// Mitsubishi GX Works2 project: a16   PLC: Q02/Q02H

PROGRAM MAIN
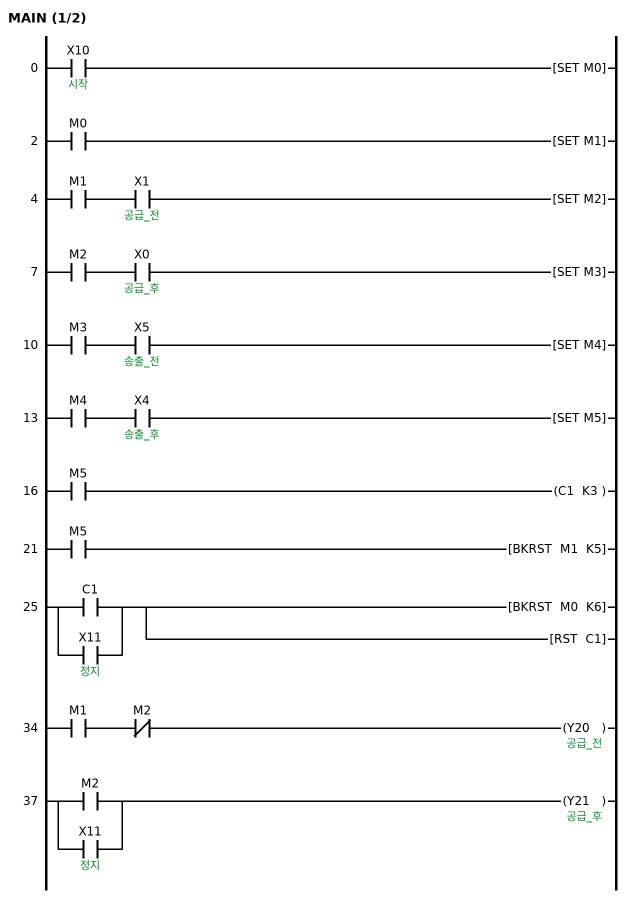
0     LD      X10  ; 시작
      SET     M0
2     LD      M0
      SET     M1
4     LD      M1
      AND     X1  ; 공급_전
      SET     M2
7     LD      M2
      AND     X0  ; 공급_후
      SET     M3
10    LD      M3
      AND     X5  ; 송출_전
      SET     M4
13    LD      M4
      AND     X4  ; 송출_후
      SET     M5
16    LD      M5
      OUT     C1 K3
21    LD      M5
      BKRST   M1 K5
25    LD      C1
      OR      X11  ; 정지
      BKRST   M0 K6
      RST     C1
34    LD      M1
      ANI     M2
      OUT     Y20  ; 공급_전
37    LD      M2
      OR      X11  ; 정지
      OUT     Y21  ; 공급_후
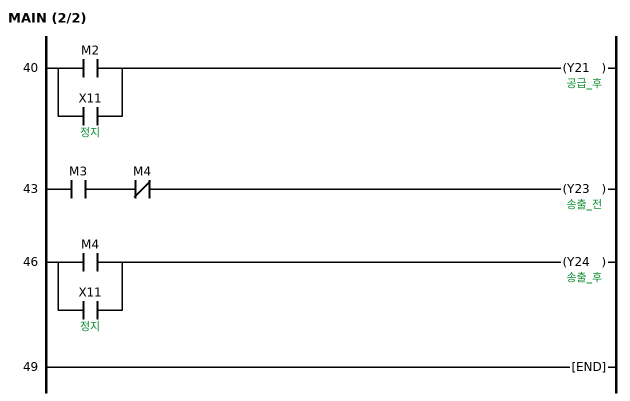
40    LD      M2
      OR      X11  ; 정지
      OUT     Y21  ; 공급_후
43    LD      M3
      ANI     M4
      OUT     Y23  ; 송출_전
46    LD      M4
      OR      X11  ; 정지
      OUT     Y24  ; 송출_후
49    END
END_PROGRAM

// device comments not shown above
X2  ; 드릴_상
X3  ; 드릴_하
X6  ; 배출_후
X7  ; 배출_전
Y22  ; 드릴_하
Y25  ; 배출_전
Y26  ; 배출_후
Y29  ; RL
Y2A  ; YL
Y2B  ; GL
